// TIA Portal project "LearningFactory_4_0_24V_Task03_CameraSSC" (V16)

(* hardware
DEVICE "ET 200SP-Station_1"  ET 200SP-Station
   slot 0: "Baugruppenträger_0"  Rack  6ES5 710-8MAx1
   slot 1: "PLC"  CPU 1512SP-1 PN  6ES7 512-1DK01-0AB0  V2.8
      slot 32768: "PROFINET"  X1
   slot 2: "DO1+2"  DQ 16x24VDC/0.5A ST  6ES7 132-6BH01-0BA0  V0.0
      slot 1: "DO1+2"  DQ 16x24VDC/0.5A ST
   slot 3: "DO3+4"  DQ 16x24VDC/0.5A ST  6ES7 132-6BH01-0BA0  V0.0
      slot 1: "DO3+4"  DQ 16x24VDC/0.5A ST
   slot 4: "DO5+6"  DQ 16x24VDC/0.5A ST  6ES7 132-6BH01-0BA0  V0.0
      slot 1: "DO5+6"  DQ 16x24VDC/0.5A ST
   slot 5: "DO7-14"  DQ 4x24VDC/2A HS  6ES7 132-6BD20-0DA0  V2.0
      slot 1: "DO7-14"  DQ 4x24VDC/2A HS
   slot 6: "DO15-22"  DQ 4x24VDC/2A HS  6ES7 132-6BD20-0DA0  V2.0
      slot 1: "DO15-22"  DQ 4x24VDC/2A HS
   slot 7: "DO23-30"  DQ 4x24VDC/2A HS  6ES7 132-6BD20-0DA0  V2.0
      slot 1: "DO23-30"  DQ 4x24VDC/2A HS
   slot 8: "DI1+2"  DI 16x24VDC ST  6ES7 131-6BH01-0BA0  V0.0
      slot 1: "DI1+2"  DI 16x24VDC ST
   slot 9: "DI3+4"  DI 16x24VDC ST  6ES7 131-6BH01-0BA0  V0.0
      slot 1: "DI3+4"  DI 16x24VDC ST
   slot 10: "DI5"  DI 8x24VDC HS  6ES7 131-6BF00-0DA0  V1.0
      slot 1: "DI5"  DI 8x24VDC HS
   slot 11: "DI6"  DI 8x24VDC HS  6ES7 131-6BF00-0DA0  V1.0
      slot 1: "DI6"  DI 8x24VDC HS
   slot 12: "AI7-10"  AI 2xU ST  6ES7 134-6FB00-0BA1  V1.0
      slot 1: "AI7-10"  AI 2xU ST
   slot 13: "End"  Server module  6ES7 193-6PA00-0AA0  V1.1
      slot 1: "End"  Server module
   slot 127: "BA 2xRJ45"  BA 2xRJ45  6ES7 193-6AR00-0AA0  V0.0
      slot 32769: "Port_1"  6ES7 193-6AR00-0AA0
      slot 32770: "Port_2"  6ES7 193-6AR00-0AA0
*)

// ===== PLC "PLC"  CPU 1512SP-1 PN =====

VAR_GLOBAL   // PLC tag table "Start_Stop"
   "IX_START" AT %I4.4 : Bool;
   "IX_STOP" AT %I4.6 : Bool;
END_VAR

VAR_GLOBAL   // PLC tag table "SSC - Camera-Station"
   "IX_SSC_RefSwitchVerticalAxis_I1" AT %I4.0 : Bool;
   "IX_SSC_RefSwitchHorizontalAxis_I2" AT %I4.1 : Bool;
   "IX_SSC_EncoderVerticalAxisImp1_B1" AT %I5.3 : Bool;
   "IX_SSC_EncoderVerticalAxisImp2_B2" AT %I5.7 : Bool;
   "IX_SSC_EncoderHorizontalAxisImp1_B3" AT %I6.3 : Bool;
   "IX_SSC_EncoderHorizontalAxisImp2_B4" AT %I6.7 : Bool;
   "QX_SSC_M1_VerticalAxisUp_Q1" AT %Q6.0 : Bool;
   "QX_SSC_M1_VerticalAxisDown_Q2" AT %Q6.1 : Bool;
   "QX_SSC_M2_HorizontalAxisClockwise_Q3" AT %Q6.3 : Bool;
   "QX_SSC_M2_HorizontalAxisCounterclockwise_Q4" AT %Q6.2 : Bool;
   "QW_SSC_PWM_Vertical_M1" AT %QW27 : Int;
   "QW_SSC_PWM_Horizontal_M2" AT %QW29 : Int;
END_VAR

DATA_BLOCK "Task03_MoveCamera_DB"   // DB1
{ S7_Optimized_Access := 'TRUE' }
VERSION : 0.1
// stored: InstanceOfName Task03_MoveCamera
"Task03_MoveCamera"
BEGIN
END_DATA_BLOCK

FUNCTION_BLOCK "Task03_MoveCamera"   // FB1, SCL
{ S7_Optimized_Access := 'TRUE' }
VERSION : 0.1
   VAR_INPUT
      Start : Bool;
      Stop : Bool;
      RefSwitchVerticalAxis : Bool;
      RefSwitchHorizontalAxis : Bool;
   END_VAR
   VAR_OUTPUT
      M1_VerticalAxisDown : Bool;
      M1_VerticalAxisUp : Bool;
      M2_HorizontalAxisClockwise : Bool;
      M2_HorizontalAxisCounterclockwise : Bool;
   END_VAR
   VAR
      R_TRIG_Start : R_TRIG;
      mem_reference_vertical : Bool;
      mem_reference_horizontal : Bool;
      IEC_Timer_Pulse : TP_TIME;
   END_VAR
BEGIN
   // Program positioning camera
   // Programm Kamerapositionierung


   //With pushbutton START move horizontal axis clockwise
   //and vertical axis down to reference position
   //Mit START-Taster Achse horizontal im Uhrzeigersinn
   //und vertikal abwärts auf Referenzposition fahren

   //Detect positive signal edge
   //Positive Signalflanke erkennen
   #R_TRIG_Start(CLK := #Start);

   IF #R_TRIG_Start.Q AND NOT #Stop THEN
       #mem_reference_horizontal := TRUE;
       #mem_reference_vertical := TRUE;
   END_IF;
   IF  #RefSwitchHorizontalAxis OR #Stop THEN
       #mem_reference_horizontal := FALSE;
   END_IF;
   IF #RefSwitchVerticalAxis  OR #Stop THEN
       #mem_reference_vertical := FALSE;
   END_IF;
   #M2_HorizontalAxisClockwise := #mem_reference_horizontal;
   #M1_VerticalAxisDown := #mem_reference_vertical;


   //With pushbutton STOP move horizontal axis counter-clockwise
   //and vertical axis up for 2 seconds
   //Mit STOP-Taster für 2 Sekunden Achse horizontal gegen Uhrzeigersinn
   //und vertikale Achse aufwärts fahren.

   //IEC-Timer TP generates pulse of 2 seconds
   //IEC-Timer TP erzeugt einen Impulse von 2 Sekunden 
   #IEC_Timer_Pulse(IN := #Stop ,
                    PT := T#2s);
   IF #Start THEN
       RESET_TIMER(#IEC_Timer_Pulse);
   END_IF;

   IF #IEC_Timer_Pulse.Q THEN
       #M1_VerticalAxisUp := TRUE;
       #M2_HorizontalAxisCounterclockwise := TRUE;
   ELSE
       #M1_VerticalAxisUp := FALSE;
       #M2_HorizontalAxisCounterclockwise := FALSE;
   END_IF;
END_FUNCTION_BLOCK

ORGANIZATION_BLOCK "Main"   // OB1, SCL, ProgramCycle
TITLE = "Main Program Sweep (Cycle)"
{ S7_Optimized_Access := 'TRUE' }
VERSION : 0.1
   VAR_INPUT
      Initial_Call : Bool;   // Initial call of this OB
      Remanence : Bool;   // =True, if remanent data are available
   END_VAR
BEGIN


   // Call subroutine MoveCamera
   // Aufruf Unterprogramm MoveCamera

   "Task03_MoveCamera_DB"(Start:="IX_START",
                          Stop:= NOT "IX_STOP",
                          RefSwitchHorizontalAxis:="IX_SSC_RefSwitchHorizontalAxis_I2",
                          RefSwitchVerticalAxis:="IX_SSC_RefSwitchVerticalAxis_I1",
                          M1_VerticalAxisDown=>"QX_SSC_M1_VerticalAxisDown_Q2",
                          M1_VerticalAxisUp=>"QX_SSC_M1_VerticalAxisUp_Q1",
                          M2_HorizontalAxisClockwise=>"QX_SSC_M2_HorizontalAxisClockwise_Q3",
                          M2_HorizontalAxisCounterclockwise=>"QX_SSC_M2_HorizontalAxisCounterclockwise_Q4");
END_ORGANIZATION_BLOCK